(* CODESYS project mqtt_client.20200326.1.project

Project tree, tasks and I/O mapping:
  Device : Changsha-Cyber-MI-linux, Changsha Cyber-MI Co., Ltd., version 3.5.10.40
    application Application
      libraries: Standard, * (System); CAA Memory, 3.5.12.0 (CAA Technical Workgroup); SysTypes2 Interfaces, 3.5.4.0 (System); CAA Net Base Services, 3.5.15.0 (CAA Technical Workgroup); CAA Types Extern, 3.5.13.0 (CAA Technical Workgroup); SysFile, 3.5.15.0 (System); MIC7001 base library, 0.80 (Cyber-MI.com); Util, 3.5.14.0 (System)
      task MainTask (cyclic, interval 10 ms, priority 10, watchdog 200 ms x 1) calls prg_mqtt
      MQTT_Client/
        Function Blocks/
          function block FB_CalculateRemainingLength [ST]
          function block FB_DecodeRemainingLength [ST]
          function block FB_MQTTClient [ST]: m_fill_subscribe_buf, m_fill_publish_buf, m_fill_connect_buf, rm_return, m_read_config
          function block FB_Random [ST]
        Structs/
          data type DUT_json
        Functions/
          function MQTTPacket_encode [ST]
          function MQTTPacket_len [ST]
          function MQTT_connect_len [ST]
          function arr2json [ST]
          function json2arr [ST]
          function get_sub_string [ST]
          function count_char_in_string [ST]
          function rm_left [ST]
      trace Trace (task MainTask): prg_main.rpm_value
      program prg_mqtt [CFC]: ACT_boot, ACT_publish, ACT_recv_proc, ACT_first_buffer, ACT_normal_buffer, ACT_running_light, proc_get_command, proc_set_command, find_key
      global variables GVL
    SoftMotion General Axis Pool
    IoDrvMIC7001 : IoDrvMIC7001, Cyber-MI, version 19.1.1
        output Application.prg_mqtt.led_run : BOOL  // LED_run
        output Application.prg_mqtt.led_err : BOOL  // LED_err
        output Application.prg_mqtt.led_usr : BOOL  // LED_usr
        unmapped channels: Ai00@C16, Ai01@C28, Ai02@C17, Ai03@C29, Ai04@C30, Ai05@C19, Ai06@C31, Ai07@C20, Ai08@C18, Ai09@D18, Ai10@D20, Ai11@D31, Ai12@D19, Ai13@D30, Ai14@D29, Ai15@D17, Ai16@D28, Ai17@D16, Ai18-Do00@C25, Ai19-Do01@C24, Ai20-Do02@C13, Ai21-Do03@C01, Ai22-Do04@C03, Ai23-Do05@C04, Ai24-Do06@C05, Ai25-Do07@C06, Ai26-Do08@C08, Ai27-Do09@C09, Ai28-Do10@C10, Ai29-Do11@C11, Ai30-Do12@D34, Ai31-Do13@D35, Ai32-Do14@D23, Ai33-Do15@D12, Ai34-Do16@D10, Ai35-Do17@D09, Ai36-Do18@D08, Ai37-Do19@D07, Ai38-Do20@D05, Ai39-Do21@D04,
          Ai40-Do22@D03, Ai41-Do23@D02, Ai42-Do24@C23, Ai43-Do25@C35, Ai44-Do26@D24, Ai45-Do27@D13, Ai46-Ao00@C22, Ai47-Ao01@D14, Ai48_Pi02, Ai49_Out5V, Ai50_VCC, Ai51_VCC_L, Ai52_VCC_R, Ai53_Pwm-i0, Ai54_Pwm-i1, Ai55_Pwm-i2, Ai56_Pwm-i3, Ai57_CPU-T, Ai58_G-x, Ai59_G-y, Ai60_G-z, Ai61-reserved, Ai62-IO-cntr, Ai63-CDS-cntr, Di00-Ai00@C16, Di01-Ai01@C28, Di02-Ai02@C17, Di03-Ai03@C29, Di04-Ai04@C30, Di05-Ai05@C19, Di06-Ai06@C31, Di07-Ai07@C20, Di08-Ai08@C18, Di09-Ai09@D18, Di10-Ai10@D20, Di11-Ai11@D31, Di12-Ai12@D19, Di13-Ai13@D30, Di14-Ai14@D29, Di15-Ai15@D17,
          Di16-Ai16@D28, Di17-Ai17@D16, Di18-Ai18@C25, Di19-Ai19@C24, Di20-Ai20@C13, Di21-Ai21@C01, Di22-Ai22@C03, Di23-Ai23@C04, Di24-Ai24@C05, Di25-Ai25@C06, Di26-Ai26@C08, Di27-Ai27@C09, Di28-Ai28@C10, Di29-Ai29@C11, Di30-Ai30@D34, Di31-Ai31@D35, Di32-Ai32@D23, Di33-Ai33@D12, Di34-Ai34@D10, Di35-Ai35@D09, Di36-Ai36@D08, Di37-Ai37@D07, Di38-Ai38@D05, Di39-Ai39@D04, Di40-Ai40@D03, Di41-Ai41@D02, Di42-Ai42@C23, Di43-Ai43@C35, Di44-Ai44@D24, Di45-Ai45@D13, Di46-Ai46@C22, Di47-Ai47@D14, Di48-Pi00@C15, Di49-Pi01@C14, Di50-Pi02@D22, Di51-Pi03@D21, Di52-reserved, Di53-reserved, Di54-reserved, Di55-reserved,
          Di56-reserved, Di57-reserved, Di58-reserved, Di59-reserved, Di60-reserved, Di61-reserved, Di62-reserved, Di63-reserved, Pi00-Di48@C15, Pi01-Di49@C14, Pi02-Di50@D22, Pi03-Di51@D21, Do00-Ai18@C25, Do01-Ai19@C24, Do02-Ai20@C13, Do03-Ai21@C01, Do04-Ai22@C03, Do05-Ai23@C04, Do06-Ai24@C05, Do07-Ai25@C06, Do08-Ai26@C08, Do09-Ai27@C09, Do10-Ai28@C10, Do11-Ai29@C11, Do12-Ai30@D34, Do13-Ai31@D35, Do14-Ai32@D23, Do15-Ai33@D12, Do16-Ai34@D10, Do17-Ai35@D09, Do18-Ai36@D08, Do19-Ai37@D07, Do20-Ai38@D05, Do21-Ai39@D04, Do22-Ai40@D03, Do23-Ai41@D02, Do24-Ai42@C23, Do25-Ai43@C35, Do26-Ai44@D24, Do27-Ai45@D13,
          Do28-Pwmi00@C33, Do29-Pwmi01@C34, Do30-Pwmi02@D25, Do31-Pwmi03@D26, PWM00@C25, PWM01@C24, PWM02@C13, PWM03@C01, PWM04@C03, PWM05@C04, PWM06@C05, PWM07@C06, PWM08@C08, PWM09@C09, PWM10@C10, PWM11@C11, PWM12@D34, PWM13@D35, PWM14@D23, PWM15@D12, PWM16@D10, PWM17@D09, PWM18@D08, PWM19@D07, PWM20@D05, PWM21@D04, PWM22@D03, PWM23@D02, PWM24@C23, PWM25@C35, PWM26@D24, PWM27@D13, PWM28-Pwmi00@C33, PWM29-Pwmi01@C34, PWM30-Pwmi02@D25, PWM31-Pwmi03@D26, PWM_I_0@C33, PWM_I_1@C34, PWM_I_2@D25, PWM_I_3@D26,
          Ao00-Ai46@C22, Ao01-Ai47@D14, ctrl_ai_raw, ctrl_adjust, ctrl_adj0, ctrl_adj1, ctrl_adj2, ctrl_adj3, disable_5V
*)

// Device/Application/MQTT_Client/Structs/DUT_json
TYPE DUT_json :
STRUCT
	key:STRING(32);
	value_dint : DINT;
	value_real : REAL;
	value_str : STRING(128);
	val_tp : UINT;  //0:  int,   1: real,    2: string
END_STRUCT
END_TYPE

// Device/Application/GVL
{attribute 'qualified_only'}

(*start of var_global for mqtt ***************************************************)
VAR_GLOBAL
	xLock_cmd : BOOL := FALSE;
	diLock_grade : DINT := 0;
	diLock_delay : DINT := 0;
	mqtt_interval : DINT := 5;  //mqtt package interval of publish to server
END_VAR

VAR_GLOBAL CONSTANT
	TYPE_DINT:UINT := 0;
	TYPE_REAL:UINT := 1;
	TYPE_STRING:UINT := 2;
END_VAR
(*end of var_global for mqtt *****************************************************)

// Device/Application/prg_mqtt
PROGRAM prg_mqtt

VAR
	FB_MQTTClient_0: FB_MQTTClient;
	
	//topic : STRING(255) := '/sys/a1SB8J9cA4L/CMI010319120011/thing/model/up_raw';
	//topic : STRING(255) := '/a1SB8J9cA4L/CMI010319120011/user/to_app';
	payload : STRING(255) := '{"RPM": 1234, "Hours": 2345}';
	
	//subscribe : STRING(255) := '/a1SB8J9cA4L/CMI010319120011/user/from_app';
	
	xPub : BOOL := FALSE;
	xSub : BOOL := FALSE;
	xBooted :BOOL := FALSE;
	
	ton_pub : ton;
	
	val_payload:ARRAY[0..32] OF dut_json;
	rpm_value : DINT := 1000;
	hours_value :REAL := 680;
	time_value : STRING;
	sn_value : STRING(128);
	lac_str:STRING(128);
	cid_str:STRING(128);
	press_value :REAL := 20.1;
	
	recv_data : ARRAY[0..32] OF DUT_json;
	old_recv_cntr:UDINT := 0;
	payload_len :INT;
	
	mqtt_first :BOOL := TRUE;
	ton_running:ton:=(pt := T#500MS);
	led_run:BOOL := FALSE;
	led_err:BOOL := FALSE;
	led_usr:BOOL := FALSE;
	pkg_id :DINT := 0;
	i :DINT;
END_VAR

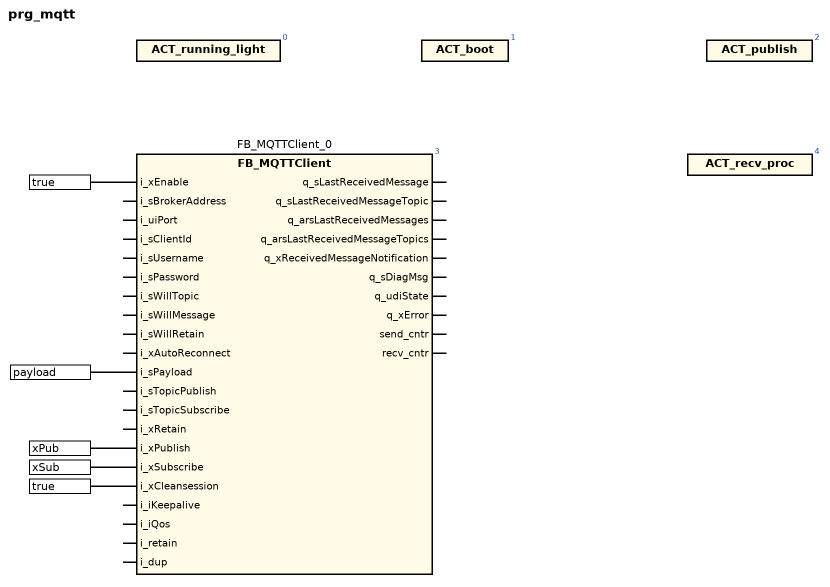
ACT_running_light();
ACT_boot();
ACT_publish();
FB_MQTTClient_0(
    i_xEnable := true,
    i_sPayload := payload,
    i_xPublish := xPub,
    i_xSubscribe := xSub,
    i_xCleansession := true); // FB_MQTTClient
ACT_recv_proc();

ACTION ACT_boot:
IF NOT xbooted THEN
	IF FB_MQTTClient_0.q_udiState = 60 THEN
		FB_MQTTClient_0.i_xSubscribe := TRUE;
		xBooted := TRUE;
	END_IF
END_IF
END_ACTION

ACTION ACT_publish:
IF FB_MQTTClient_0.q_udiState <> 60 THEN   //not ready, return and wait
	xPub := FALSE;
	RETURN;
END_IF

IF mqtt_first THEN
	mqtt_first := FALSE;
	ACT_first_buffer();
	xPub := TRUE;
	RETURN;
END_IF

ton_pub(in := NOT ton_pub.Q, pt := ANY_TO_TIME(gvl.mqtt_interval*1000));   // second to ms
IF ton_pub.Q THEN
	ACT_normal_buffer();
	xPub := TRUE;
ELSE
	xPub := FALSE;
END_IF
END_ACTION

ACTION ACT_recv_proc:
(*
	cmd:  	set, get          			//命令字, set:设置参数或者执行命令，  get：点播数据或参数
	act:  	lock, unlock, reboot		//动作类型
	grade:  1, 2, 3, 4					//动作级别
	delay:  0, 60, 3600					//延迟时间,单位： 秒
*)

IF old_recv_cntr = FB_MQTTClient_0.recv_cntr THEN  //no new message
	RETURN;
END_IF
old_recv_cntr := FB_MQTTClient_0.recv_cntr;

payload_len := json2arr(json := FB_MQTTClient_0.q_sLastReceivedMessage, pArr := ADR(recv_data), max_len := 32);
IF payload_len = 0 THEN
	RETURN;
END_IF

i := find_key(key := 'cmd');
IF i >= 0 AND recv_data[i].val_tp = GVL.TYPE_STRING THEN 
	IF  recv_data[i].value_str = 'get' THEN
		proc_get_command();
	ELSIF recv_data[i].value_str = 'set' THEN
		proc_set_command();
	END_IF
END_IF
END_ACTION

ACTION ACT_first_buffer:

val_payload[0].key := 'sn';
val_payload[0].val_tp := GVL.TYPE_STRING;
IF MIC7001_base.read_sn(ADR(sn_value)) THEN
	val_payload[0].value_str := sn_value;
ELSE
	val_payload[0].value_str := 'SN Error';
END_IF

val_payload[1].key := 'lac';
val_payload[1].val_tp := GVL.TYPE_STRING;

val_payload[2].key := 'cid';
val_payload[2].val_tp := GVL.TYPE_STRING;

IF MIC7001_base.read_location(lac := ADR(lac_str), ci := ADR(cid_str)) THEN
	val_payload[1].value_str := lac_str; 
	val_payload[2].value_str := cid_str; 
ELSE
	val_payload[1].value_str := 'lac_error'; 
	val_payload[2].value_str := 'cid_error'; 
END_IF

payload := arr2json(arr := val_payload, num := 3);
END_ACTION

ACTION ACT_normal_buffer:

val_payload[0].key := 'rpm';
val_payload[0].val_tp := GVL.TYPE_DINT; 
rpm_value := rpm_value + 1;
IF rpm_value > 2200 THEN
	rpm_value := 1000;
END_IF
val_payload[0].value_dint := rpm_value; 

val_payload[1].key := 'hour_all';
val_payload[1].val_tp := GVL.TYPE_REAL;
hours_value := hours_value + 5.0/3600;
val_payload[1].value_real := hours_value; 

val_payload[2].key := 'power';
val_payload[2].val_tp := GVL.TYPE_REAL;  
val_payload[2].value_real := ANY_TO_REAL(rpm_value)/10.0 - 39.0; 

val_payload[3].key := 'press';
val_payload[3].val_tp := GVL.TYPE_REAL;  
press_value := press_value + 0.001;
IF press_value > 35 THEN
	press_value := 20;
END_IF
val_payload[3].value_real := press_value; 

val_payload[4].key := 'fuel_all';
val_payload[4].val_tp := GVL.TYPE_REAL;  
val_payload[4].value_real := ANY_TO_REAL(hours_value)*13.2; 

val_payload[5].key := 'pkg_id';
val_payload[5].val_tp := GVL.TYPE_DINT; 
pkg_id := pkg_id + 1;
val_payload[5].value_dint := pkg_id; 

payload := arr2json(arr := val_payload, num := 6);
END_ACTION

ACTION ACT_running_light:
ton_running(in := NOT ton_running.Q);
IF ton_running.Q THEN
	led_run := NOT led_run;
	led_usr := FALSE;
END_IF

IF FB_MQTTClient_0.q_udiState <> 60 THEN
	led_usr := TRUE;
END_IF
END_ACTION

ACTION proc_get_command:
(*
	cmd:  	get  	//命令字, get：点播数据或参数
	rpm:  	15		//点播转速， 上传15次
	press:  0		//点播压力， 持续上传
	fuel_all: 1	  	//点播总油耗，上传一次 					
*)
END_ACTION

ACTION proc_set_command:
(*
	cmd:  	set  	          	//命令字, set:设置参数或者执行命令，  get：点播数据或参数
	interval:	15				//设置上传间隔： 15秒
	act:  	lock, unlock		//锁机动作类型
	grade:  1, 2, 3, 4			//动作级别
	delay:  0, 60, 3600			//延迟时间,单位： 秒
*)

// check lock command 
i := find_key(key := 'act');
IF i >= 0 AND recv_data[i].val_tp = GVL.TYPE_STRING  THEN
	IF recv_data[i].value_str = 'lock' THEN
		gvl.xlock_cmd := TRUE;
	ELSIF recv_data[i].value_str = 'unlock' THEN
		gvl.xlock_cmd := FALSE;
	END_IF
END_IF

i := find_key(key := 'grade');
IF i >= 0 AND recv_data[i].val_tp = GVL.TYPE_DINT THEN
	gvl.diLock_grade := recv_data[i].value_dint;
END_IF

i := find_key(key := 'delay');
IF i >= 0 AND recv_data[i].val_tp = GVL.TYPE_DINT THEN
	gvl.diLock_delay := recv_data[i].value_dint;
END_IF

i := find_key(key := 'interval');
IF i >= 0 AND recv_data[i].val_tp = GVL.TYPE_DINT THEN
	gvl.mqtt_interval := recv_data[i].value_dint;
END_IF
END_ACTION

METHOD find_key : dint
VAR_INPUT
	key :STRING(32);
END_VAR
VAR
	i :UINT;
END_VAR
find_key := -1;

FOR i := 0 TO payload_len-1 DO
	IF key = recv_data[i].key THEN
		find_key := i;
		RETURN;
	END_IF
END_FOR

RETURN; // not find,  return -1
END_METHOD

END_PROGRAM

// Device/Application/MQTT_Client/Function Blocks/FB_MQTTClient
(*  mqtt client for MIC7001
    by zhoujihui@gmail.com
*)
FUNCTION_BLOCK FB_MQTTClient
VAR_INPUT
	// Enables the Function block, The rising Edge of this Input automatically connects to the MQTT Broker - Standard: TRUE
	i_xEnable: BOOL := TRUE;
	// IP-Address (example: 192.168.178.101) or Webaddress (www.mqtt-dashboard.com) of the MQTT-Broker
	i_sBrokerAddress: STRING(255) := '47.107.240.29';
	// Port of the MQTT-Broker - Standard: 1883
	i_uiPort: UINT := 1883;
	// clientId
	i_sClientId: STRING(255) := 'MIC7001 client Id';
	// Optional Username if required
	i_sUsername: STRING(255) := '';
	// Optional Password if required
	i_sPassword: STRING(255) := '';
	// Last Will Topic if required (Automatically enables Will Message if changed) - otherwise leave untouched
	i_sWillTopic: STRING(255) := '';
	// Last Will Message if required - otherwise leave untouched
	i_sWillMessage: STRING(255) := '';
	// Retain Last Will Message, if required Standard: FALSE - otherwise leave untouched 
	i_sWillRetain: BOOL := FALSE;	
	// Automatically try to reconnect after an Exception - Standard: TRUE
	i_xAutoReconnect: BOOL := TRUE;
	// PayLoad to Publish
	i_sPayload: STRING(255) := '';
	// Topic to Publish to
	i_sTopicPublish: STRING(255) := '/MIC7001/without/config/files';
	// Topic to Subscribe
	i_sTopicSubscribe: STRING(255) := '';
	// Retain Flag Forces the Broker to Retain the Last Mesage - Standard: TRUE
	i_xRetain: BOOL := TRUE;
	// Publish the Payload to the Topic of the MQTT-Broker
	i_xPublish: BOOL:=FALSE;
	// Subscribe to the Topic given to the Input i_sTopicSubscribe
	i_xSubscribe: BOOL:=FALSE;
	// clean session
	i_xCleansession : BOOL := FALSE;
	// keep alive
	i_iKeepalive :INT := 60000;
	// QoS of publish packet
	i_iQos : BYTE := 0;
	// retain
	i_retain : BOOL := FALSE;
	// dup
	i_dup :BOOL := FALSE;
	
END_VAR
VAR_OUTPUT
	// Message Received from a subsribed Topic
	q_sLastReceivedMessage: STRING(255);
	// Topic Message Received
	q_sLastReceivedMessageTopic: STRING(255);	
	// Last 25 Received Messages
	q_arsLastReceivedMessages: STRING(255);
	// Last 25 Topics Received
	q_arsLastReceivedMessageTopics: STRING(255);	
	// Message Received Notification
	q_xReceivedMessageNotification: BOOL;
	// Diag Message
	q_sDiagMsg: STRING(255);
	// Current State of the Function Block
	q_udiState: UDINT;
	// Error Flag
	q_xError: BOOL;
	//publish message counter
	send_cntr :UDINT := 0;
	//received message counter
	recv_cntr: UDINT := 0;
END_VAR
VAR
	R_TRIG_Enable: R_TRIG;

	diResult: CAA.SIZE;
	IFB_CalculateRemainingLength: FB_CalculateRemainingLength;
	IFB_Random: ARRAY[0..9] OF FB_Random;
	wKeepAlive: WORD := 0;
	IoCtlParameter : DINT := 1;

	R_TRIG_Publish: R_TRIG;
	R_TRIG_Subscribe: R_TRIG;

	uiYear:UINT;
	uiMonth: UINT;
	uiDay: UINT;
	uiHour: UINT;
	uiMinute: UINT;
	uiSecond: UINT;
	
	TON_TimeOut: ton;
	wTimeOutValue: WORD;
	udiLastState: UDINT;
	
	xResultDisconnect: BOOL;
	QI: INT;
	
	iIndexCount: INT;
	wPacketIdentifierCount: WORD :=0;
	uiPayLoadLength: uint;
	
	xPublish: BOOL;
	xSubscribe: BOOL;
	
	i: INT;

	hSock:RTS_IEC_HANDLE;
	pSock_create_rst: POINTER TO RTS_IEC_RESULT;
	pSock_recv_rst: POINTER TO RTS_IEC_RESULT;
	pSock_send_rst: POINTER TO RTS_IEC_RESULT;

	ui_rc_disconnect : UDINT;
	pInaddr:POINTER TO STRING;
	
	tcp_client : NBS.TCP_Client;
	tcp_connection : CAA.HANDLE;
	tcp_send : NBS.TCP_Write;
	tcp_recv : NBS.TCP_Read;
	s_send_buf : ARRAY[0..999] OF BYTE;
	s_recv_buf : ARRAY[0..999] OF BYTE;
	udi_time_out : UDINT;
	server_ip : NBS.IP_ADDR;
	buf_size : CAA.size;
	recv_len : INT;

	header :BYTE ; 
	bytes_len_rem : INT;
	length_topic : INT;
	recv_qos : BYTE := 0;
	id_msb : BYTE;
	id_lsb : BYTE;
	hFile: RTS_IEC_HANDLE;
	udiOpenError: RTS_IEC_RESULT;
	udiReadError: RTS_IEC_RESULT;
	str_size: __XWORD;
	udiByteRead: LWORD;	
	str_temp:STRING(255);
	error_cntr : DINT := 0;
END_VAR


R_TRIG_Enable(CLK:=i_xEnable);
R_TRIG_Publish(CLK:=i_xPublish);
R_TRIG_Subscribe(CLK:=i_xSubscribe);

IF (R_TRIG_Publish.Q) THEN
	xPublish:=TRUE;
END_IF

IF (R_TRIG_Subscribe.Q) THEN
	xSubscribe:=TRUE;
END_IF

CASE q_udiState OF
//0: Wait for Enable
0: 	wTimeOutValue:=0;
	
	IF (NOT q_xError) THEN	
		q_sDiagMsg:='Wait for Enable';
	END_IF
	
	IF (i_xEnable OR (i_xAutoReconnect AND q_xError)) THEN
		IF m_read_config() THEN
			q_xError := FALSE;
			q_udiState:=5;
			tcp_client(xEnable := FALSE);
			server_ip.sAddr := i_sBrokerAddress;
			tcp_client.xEnable := TRUE;			
			q_sDiagMsg:='Creating TCP connect';
		ELSE
			q_xError := TRUE;
			q_sDiagMsg:='Failed reading config files';
			q_udiState:=99;
		END_IF
		
	END_IF

5:  
	IF tcp_client.xActive THEN
		q_udiState := 15;
		q_sDiagMsg:='Initialize send-Buffer';
	END_IF
	
	wTimeOutValue:=3000;
	IF (TON_TimeOut.Q) THEN
		q_udiState:=0;	
	END_IF		

//15: Initialize OutBuffer
15:
	buf_size := m_fill_connect_buf();
	IF buf_size > 0 THEN
		tcp_send.szSize := buf_size; 
		tcp_send(xExecute := FALSE);
		tcp_send.xExecute := TRUE;
		tcp_recv.xEnable := TRUE;
		
		q_udiState:=20;
		q_sDiagMsg:='Connect to MQTT-Broker';
	ELSE
		q_xError := TRUE;
		q_sDiagMsg:='Send buffer is Error.';
		q_udiState:=0;
	END_IF
	
//20: Send Connect	
20:		
	wTimeOutValue:=1000;
	tcp_recv(hConnection := tcp_connection, szSize := 1024, pData := ADR(s_recv_buf));
	IF tcp_recv.xReady  THEN
		q_udiState:= 30;
	END_IF
	
	IF (TON_TimeOut.Q) THEN
		q_udiState:=0;	
		q_xError := TRUE;
		q_sDiagMsg:='Connecting to MQTT-Broker (MQTT Control Packet) Timed out';
	END_IF
//30: Analyze CONNACK
30:	q_sDiagMsg:='Analyze connack';
	wTimeOutValue:=0;
	
	IF (s_recv_buf[0] = 32 AND s_recv_buf[3] = 0) THEN
		q_udiState := 60;
	ELSE
		//Return code repsone (2nd Byte): 
		//0: Connection Accepted
		//1: Connection Refused, unacceptable protocol version
		IF (s_recv_buf[3] = 1) THEN
			q_sDiagMsg:='Connection Refused, unacceptable protocol version';
		END_IF
		//2: Connection Refused, identifier rejected
		IF (s_recv_buf[3] = 2) THEN
			q_sDiagMsg:='Connection Refused, identifier rejected';
		END_IF
		//3: Connection Refused, Server unavailable
		IF (s_recv_buf[3] = 3) THEN
			q_sDiagMsg:='Connection Refused, Server unavailable';
		END_IF		
		//4: Connection Refused, bad Username or passworrd
		IF (s_recv_buf[3] = 4) THEN
			q_sDiagMsg:='Connection Refused, bad Username or password';
		END_IF	
		//5: Connection Refused, not autorized
		IF (s_recv_buf[3] = 5) THEN
			q_sDiagMsg:='Connection Refused, not autorized';
		END_IF	
		q_xError := TRUE;
		q_udiState := 90;	
	END_IF
	
//60: Wait for Publish or Disconnect (Enable low)
60:	q_sDiagMsg:='Wait for Publish or Subscribe or Disconnect (Enable low)';
	wTimeOutValue:=0;
	q_xReceivedMessageNotification:= FALSE;

	IF (xPublish) THEN
		xPublish:=FALSE;
		q_udiState := 70;	
	END_IF
	IF (xSubscribe) THEN
		xSubscribe:=FALSE;
		q_udiState := 65;	
	END_IF
	IF (NOT i_xEnable) THEN
		q_udiState := 80;	
	END_IF
	
	tcp_recv(hConnection := tcp_connection, szSize := 1024, pData := ADR(s_recv_buf));
	IF tcp_recv.szCount > 2 THEN
		header := s_recv_buf[0];
		IF header.5 AND header.4 AND tcp_recv.szCount < 1024 THEN   // publish:  0x30
			q_xReceivedMessageNotification:= TRUE;
			diResult := tcp_recv.szCount;
			q_udiState := 63;
			
		END_IF	
	END_IF
	
//Analyze Publish Message from Broker
63: q_sDiagMsg:='Analyze Publish Message from Broker';
	wTimeOutValue:=0;

	IFB_CalculateRemainingLength(wNumberOfBytes:=ANY_TO_WORD(diResult-2));
	bytes_len_rem := IFB_CalculateRemainingLength.iNumberOfBytesRemianingLengthField;
	length_topic := BYTE_TO_INT(s_recv_buf[bytes_len_rem+1])*256 + s_recv_buf[bytes_len_rem+2];
	IF length_topic > 128 THEN
		q_udiState := 60;
		RETURN;	
	END_IF
	
	uiPayLoadLength:=ANY_TO_UINT(diResult - length_topic - 1 - bytes_len_rem - 2);
	header := s_recv_buf[0];
	
	recv_qos := 0;
	IF header.1 OR header.2 THEN //Qos > 0
		uiPayLoadLength :=  uiPayLoadLength - 2;  //remove 2bytes of packet Id
		IF header.1 THEN
			recv_qos := 1;
		ELSIF header.2 THEN
			recv_qos := 2;
		END_IF	

		id_msb := s_recv_buf[1+bytes_len_rem + 2 + length_topic];
		id_lsb := s_recv_buf[1+bytes_len_rem + 2 + length_topic+1];
	END_IF
	
	mem.MemFill(ADR(q_sLastReceivedMessage),255,0);
	mem.MemFill(ADR(q_sLastReceivedMessageTopic),255,0);
	MEM.MemMove(ADR(s_recv_buf[diResult-uiPayLoadLength]),ADR(q_sLastReceivedMessage),uiPayLoadLength);
	MEM.MemMove(ADR(s_recv_buf[IFB_CalculateRemainingLength.iNumberOfBytesRemianingLengthField+3]),ADR(q_sLastReceivedMessageTopic),length_topic);
	
	q_arsLastReceivedMessageTopics:=q_sLastReceivedMessageTopic;
	q_arsLastReceivedMessages:=q_sLastReceivedMessage;
	
	diResult:=0;
	recv_cntr := recv_cntr + 1;
	IF recv_qos = 0 THEN
		q_udiState := 60;
	ELSIF recv_qos = 1 THEN
		
		s_send_buf[0] := 16#40;  //type: puback
		s_send_buf[1] := 2;
		s_send_buf[2] := id_msb;
		s_send_buf[3] := id_lsb;
		tcp_send(xExecute := FALSE);
		tcp_send.xExecute := TRUE;
		tcp_send.szSize := 4;
		q_udiState := 64; // send ack
		wTimeOutValue:=1000;
		q_sDiagMsg:='Send ack to broker';
	ELSE  // qos = 2, not support yet
		q_udiState := 60;
	END_IF	

64:
	IF tcp_send.xDone THEN
		q_udistate := 60;
	END_IF
//65: Subscribe to Topic
65: q_sDiagMsg:='Subscribe to Topic';
	wTimeOutValue:=1000;
	
	buf_size := m_fill_subscribe_buf();
	IF buf_size > 0 THEN
		tcp_send.szSize := buf_size; 
		tcp_send(xExecute := FALSE);
		tcp_send.xExecute := TRUE;
		tcp_recv.xEnable := TRUE;
		q_udiState:=66;	
	ELSE
		q_xError := TRUE;
		q_sDiagMsg:='Subscribe buffer is Error.';
		q_udiState:=0;
	END_IF
	
	tcp_recv(hConnection := tcp_connection, szSize := 1024, pData := ADR(s_recv_buf));
	IF tcp_recv.xDone THEN 
		q_udiState:=66;	
	END_IF	
	IF (TON_TimeOut.Q) THEN
		q_udiState:=90;	
		q_xError := TRUE;
		q_sDiagMsg:='Subscribe (MQTT Control Packet) Timed out';
	END_IF	
	
//66: Wait for SUBACK from Broker
66: //diResult := SysSockRecv(hSocket := hSock,pbyBuffer:=ADR(inBuffer),diBufferSize:=500,diFlags:=0, ADR(pSock_recv_rst));
	q_sDiagMsg:='Wait for SUBACK from Broker';
	wTimeOutValue:=1000;
	tcp_recv(hConnection := tcp_connection, szSize := 1024, pData := ADR(s_recv_buf));
	IF tcp_recv.szCount > 0 THEN
		q_udiState:=67;	
		diResult:=0;
	END_IF
	IF (TON_TimeOut.Q) THEN
		q_udiState:=90;	
		q_xError := TRUE;
		q_sDiagMsg:='Waiting for "Suback" from MQTT-Broker Timed out';
	END_IF

//67: Analyze SUBACK
67:	q_sDiagMsg:='Analyze SUBACK';
	wTimeOutValue:=0;
	tcp_recv(hConnection := tcp_connection, szSize := 1024, pData := ADR(s_recv_buf));
	recv_len := ANY_TO_INT(tcp_recv.szCount);
	IF (s_recv_buf[recv_len-1] < 16#80) THEN
		q_udiState := 60;
		diResult:=0;
	ELSE	
		q_udiState:=90;	
		q_xError := TRUE;
		q_sDiagMsg:='Suback Message reported Failure (Return code 0x80)';
	END_IF
	
//70: Publish Message
70: 
	buf_size := m_fill_publish_buf();

	IF buf_size > 0 THEN
		tcp_send.szSize := buf_size; 
		tcp_send(xExecute := FALSE);
		tcp_send.xExecute := TRUE;
		tcp_recv.xEnable := TRUE;
		q_sDiagMsg:='Publish Message';
		wTimeOutValue:=1000;		
		q_udiState:=75;	
	END_IF
	
75:	
	IF (tcp_send.xDone > 0) THEN 
		q_udiState:=60;	
		send_cntr := send_cntr + 1;
	END_IF	
	IF (TON_TimeOut.Q) THEN
		q_udiState:=90;	
		q_xError := TRUE;
		q_sDiagMsg:='Publishing Message (MQTT Control Packet) Timed out';
	END_IF

//80: Send "Disconnect"
80: s_send_buf[0] := 224;		//MQTT Control Packet Type
	s_send_buf[1] := 0;			//Remaining Length (0)
	tcp_send.szSize := 2;
	tcp_send(xExecute := FALSE);
	tcp_send.xExecute := TRUE;
	
	q_sDiagMsg:='Send Disconnect notification to server';
	wTimeOutValue:=1000;
	q_udiState:=85;

85:	
	IF (tcp_send.xDone) THEN 
		diResult:=0;
		q_udiState:=90;	
	END_IF	
	IF (TON_TimeOut.Q) THEN
		q_udiState:=90;	
		q_xError := TRUE;
		q_sDiagMsg:='Sending Disconnect to MQTT-Broker Timed out';
	END_IF	

//90: Disconnect Socket
90:	tcp_client.xEnable := FALSE;
	IF (NOT q_xError) THEN
		q_sDiagMsg:='Close TCP Socket';
	END_IF
	wTimeOutValue:=1000;
	IF (ui_rc_disconnect = 0) THEN 
		q_udiState:=0;	
	END_IF	
	IF (TON_TimeOut.Q) THEN
		q_udiState:=0;	
		q_xError := TRUE;
		q_sDiagMsg:='Closing TCP-Socket  Timed out';
	END_IF	

99: //error
	wTimeOutValue:=5000;
	IF (TON_TimeOut.Q) THEN
		q_udiState:=0;	
		q_xError := TRUE;
		q_sDiagMsg:='Error status Timed out';
	END_IF	
END_CASE

TON_TimeOut(IN:=(udiLastState=q_udiState) AND (wTimeOutValue <> 0) ,PT:=WORD_TO_TIME(wTimeOutValue));
udiLastState:=q_udiState;

IF q_udiState >= 5 THEN
	tcp_client(xEnable := TRUE, ipAddr := server_ip, uiPort := i_uiPort , udiTimeOut := 0, hConnection => tcp_connection);
	IF tcp_connection > 0 THEN
		tcp_send(udiTimeOut := udi_time_out, hConnection := tcp_connection, pData := ADR(s_send_buf));
	END_IF
END_IF

METHOD m_fill_subscribe_buf : CAA.SIZE
VAR_INPUT
END_VAR

VAR
	i : INT;
	ui_subscribe_len:INT;
	ui_mqtt_msg_len:INT;
	ptr : INT := 0;
	rem_len :INT := 0;
	packet_len : CAA.SIZE := 0;
	rc :INT := 0;
	
	flag :BYTE := 0;
END_VAR
m_fill_subscribe_buf := 0;

ui_subscribe_len := (LEN(i_sTopicSubscribe));

rem_len := ui_subscribe_len + 2 + 2 + 1;  //packet id: 2bytes,  length: 2bytes, QoS: 1byte 
packet_len := MQTTPacket_len(rem_len);

IF packet_len > SIZEOF(s_send_buf) THEN
	m_fill_subscribe_buf := 0;
	RETURN;
END_IF

ptr := 0;
// Header Flag. subscribe command.
flag := 16#82;

IF i_dup THEN
	flag := flag + 8;
END_IF

s_send_buf[ptr] := flag;  ptr := ptr + 1;

// Msg Len.
rc := MQTTPacket_encode(ADR(s_send_buf[ptr]), rem_len);   ptr := ptr + rc;

wPacketIdentifierCount:=wPacketIdentifierCount + 1;
IF (wPacketIdentifierCount = 0) THEN
	wPacketIdentifierCount:=1;
END_IF

// packet id	
s_send_buf[ptr] := UINT_TO_BYTE(wPacketIdentifierCount / 256); ptr := ptr + 1;
s_send_buf[ptr] := UINT_TO_BYTE(wPacketIdentifierCount MOD 256); ptr := ptr + 1;

// topic Length.
s_send_buf[ptr] := UINT_TO_BYTE(ui_subscribe_len / 256); ptr := ptr + 1;
s_send_buf[ptr] := UINT_TO_BYTE(ui_subscribe_len MOD 256); ptr := ptr + 1;

//topic subscribe
FOR i:=0 TO ui_subscribe_len-1 DO
	s_send_buf[ptr] := i_sTopicsubscribe[i]; ptr := ptr + 1;
END_FOR	

s_send_buf[ptr] := i_iQos;

m_fill_subscribe_buf := packet_len;
END_METHOD

METHOD m_fill_publish_buf : CAA.SIZE
VAR_INPUT
END_VAR

VAR
	i : INT;
	ui_client_id_len : INT;
	ui_topic_len :INT;
	ui_payload_len:INT;
	ui_mqtt_msg_len:INT;
	ptr : INT := 0;
	rem_len :INT := 0;
	packet_len : CAA.size := 0;
	rc :INT := 0;
	packet_id : UINT := 1;
	flag :BYTE := 0;
END_VAR
m_fill_publish_buf := 0;

ui_topic_len := (LEN(i_sTopicPublish));
ui_payload_len := (LEN(i_sPayload));

rem_len := ui_topic_len + 2 + ui_payload_len;
IF i_iQos > 0 THEN
	rem_len := rem_len + 2;  // add 2 bytes packet Id
END_IF

packet_len := MQTTPacket_len(rem_len);

IF packet_len > SIZEOF(s_send_buf) THEN
	m_fill_publish_buf := 0;
	RETURN;
END_IF

ptr := 0;
// Header Flag. Publish command.
flag := 16#30;  //publish
IF i_retain THEN
	flag := flag + 1;
END_IF

IF i_iQos > 0 AND i_iQos < 3 THEN
	flag := flag + i_iQos*2;
ELSE
	i_dup := 0;
END_IF

IF i_dup THEN
	flag := flag + 8;
END_IF

s_send_buf[ptr] := flag;  ptr := ptr + 1;

// Msg Len.
rc := MQTTPacket_encode(ADR(s_send_buf[ptr]), rem_len);   ptr := ptr + rc;

//topic
IF ui_topic_len > 0 THEN
	// topic Length.
	s_send_buf[ptr] := UINT_TO_BYTE(ui_topic_len / 256); ptr := ptr + 1;
	s_send_buf[ptr] := UINT_TO_BYTE(ui_topic_len MOD 256); ptr := ptr + 1;
	
	// topic
	FOR i:=0 TO ui_topic_len-1 DO
		s_send_buf[ptr] := i_sTopicPublish[i]; ptr := ptr + 1;
	END_FOR	
END_IF

IF i_iQos > 0 THEN
	wPacketIdentifierCount:=wPacketIdentifierCount + 1;
	IF (wPacketIdentifierCount = 0) THEN
		wPacketIdentifierCount:=1;
	END_IF
	s_send_buf[ptr] := UINT_TO_BYTE(wPacketIdentifierCount / 256); ptr := ptr + 1;
	s_send_buf[ptr] := UINT_TO_BYTE(wPacketIdentifierCount MOD 256); ptr := ptr + 1;
END_IF

//payload
IF ui_payload_len > 0 THEN
	// payload,  no length needed
	FOR i:=0 TO ui_payload_len-1 DO
		s_send_buf[ptr] := i_spayload[i]; ptr := ptr + 1;
	END_FOR	
END_IF

m_fill_publish_buf := packet_len;
END_METHOD

METHOD m_fill_connect_buf : CAA.SIZE
VAR_INPUT
END_VAR

VAR
	ui_client_id_len : INT;	
	ui_username_len : INT;
	ui_password_len : INT;
	ui_will_topic_len : INT;
	ui_will_msg_len : INT;
	ptr:INT := 0;  
	remaining_len :INT;
	packet_len :CAA.SIZE;
	rc :INT;
	flag : BYTE := 0;
END_VAR
m_fill_connect_buf := 0;

ui_client_id_len := (LEN(i_sclientid));
ui_username_len := (LEN(i_sUsername));
ui_password_len := (LEN(i_sPassword));
ui_will_topic_len := (len(i_sWillTopic));
ui_will_msg_len := (len(i_sWillMessage));

remaining_len := MQTT_connect_len(ui_client_id_len, ui_will_topic_len, ui_will_msg_len, ui_username_len, ui_password_len);
packet_len := MQTTPacket_len(remaining_len);

IF packet_len > SIZEOF(s_send_buf) THEN
	m_fill_connect_buf := 0;
	RETURN;
END_IF

ptr := 0;

// Header Flag. Connect command.
s_send_buf[ptr] := 16#10; ptr := ptr + 1;

// Msg Len.
rc := MQTTPacket_encode(ADR(s_send_buf[ptr]), remaining_len);   ptr := ptr + rc;


// Protocal Name Length.
s_send_buf[ptr] := 16#00; ptr := ptr + 1;
s_send_buf[ptr] := 16#04; ptr := ptr + 1;
// Protocal Name.
s_send_buf[ptr] := 16#4D; ptr := ptr + 1;
s_send_buf[ptr] := 16#51; ptr := ptr + 1;
s_send_buf[ptr] := 16#54; ptr := ptr + 1;
s_send_buf[ptr] := 16#54; ptr := ptr + 1;
// Version.
s_send_buf[ptr] := 16#04; ptr := ptr + 1;

// Connect Flags.
flag := 0;
IF i_xCleansession THEN
	flag := flag + 16#02;
END_IF

IF ui_username_len > 0 THEN
	flag := flag + 16#80;
END_IF

IF ui_password_len > 0 THEN
	flag := flag + 16#40;
END_IF

s_send_buf[ptr] := flag;  ptr := ptr + 1;

// Keep Alive.
s_send_buf[ptr] := INT_TO_BYTE(i_iKeepalive / 256); ptr := ptr + 1;
s_send_buf[ptr] := INT_TO_BYTE(i_iKeepalive MOD 256); ptr := ptr + 1;

// Client ID Length.
s_send_buf[ptr] := INT_TO_BYTE(ui_client_id_len / 256); ptr := ptr + 1;
s_send_buf[ptr] := INT_TO_BYTE(ui_client_id_len MOD 256); ptr := ptr + 1;
// Client ID.
FOR i:=0 TO ui_client_id_len-1 DO
	s_send_buf[ptr] := i_sClientId[i]; ptr := ptr + 1;
END_FOR

IF ui_will_topic_len > 0 THEN
	// will topic Length.
	s_send_buf[ptr] := INT_TO_BYTE(ui_will_topic_len / 256); ptr := ptr + 1;
	s_send_buf[ptr] := INT_TO_BYTE(ui_will_topic_len MOD 256); ptr := ptr + 1;
	// will topic.
	FOR i:=0 TO ui_will_topic_len-1 DO
		s_send_buf[ptr] := i_sWilltopic[i]; ptr := ptr + 1;
	END_FOR	
END_IF

IF ui_will_msg_len > 0 THEN
	// will message Length.
	s_send_buf[ptr] := INT_TO_BYTE(ui_will_msg_len / 256); ptr := ptr + 1;
	s_send_buf[ptr] := INT_TO_BYTE(ui_will_msg_len MOD 256); ptr := ptr + 1;
	// will message.
	FOR i:=0 TO ui_will_msg_len-1 DO
		s_send_buf[ptr] := i_sWillmessage[i]; ptr := ptr + 1;
	END_FOR	
END_IF

IF ui_username_len > 0 THEN
	// will message Length.
	s_send_buf[ptr] := INT_TO_BYTE(ui_username_len / 256); ptr := ptr + 1;
	s_send_buf[ptr] := INT_TO_BYTE(ui_username_len MOD 256); ptr := ptr + 1;
	// username
	FOR i:=0 TO ui_username_len-1 DO
		s_send_buf[ptr] := i_susername[i]; ptr := ptr + 1;
	END_FOR	
END_IF

IF ui_password_len > 0 THEN
	// will message Length.
	s_send_buf[ptr] := INT_TO_BYTE(ui_password_len / 256); ptr := ptr + 1;
	s_send_buf[ptr] := INT_TO_BYTE(ui_password_len MOD 256); ptr := ptr + 1;
	// password
	FOR i:=0 TO ui_password_len-1 DO
		s_send_buf[ptr] := i_spassword[i]; ptr := ptr + 1;
	END_FOR	
END_IF


m_fill_connect_buf := packet_len;
END_METHOD

METHOD PRIVATE rm_return : string(255)
VAR_INPUT
	str_in:STRING(255);
END_VAR

VAR
	str_rc:string(255);
	length:INT;
END_VAR
str_rc := str_in;

length := len(str_rc);
IF str_rc[length-1] = 10 THEN   // $N
	str_rc := left(str_rc, length-1);
END_IF

length := len(str_rc);
IF str_rc[length-1] = 10 THEN   // $N
	str_rc := left(str_rc, length-1);
END_IF

length := len(str_rc);
IF str_rc[length-1] = 10 THEN   // $N
	str_rc := left(str_rc, length-1);
END_IF

length := len(str_rc);
IF str_rc[length-1] = 10 THEN   // $N
	str_rc := left(str_rc, length-1);
END_IF

rm_return := str_rc;
END_METHOD

METHOD m_read_config : bool
VAR_INPUT
END_VAR
m_read_config := FALSE;

hFile := sysfileopen(szFile := '/userapp/mqtt_server.txt', am := sysfile.AM_READ, pResult:= ADR(udiOpenError));
IF hFile = RTS_INVALID_HANDLE THEN
	RETURN;
END_IF

//文件存在，开始读取内容
sysfile.SysFileSetPos(hFile:=hFile, ulOffset := 0);
FOR i := 0 TO 255 DO  str_temp[i] := 0; END_FOR
udiByteRead := sysfile.SysFileRead(hfile := hFile,pbyBuffer := ADR(str_temp), ulSize := 250, pResult := ADR(udiReadError));
str_temp := rm_return(str_temp);
IF udiByteRead > 7 THEN  
	i_sBrokerAddress := str_temp;
END_IF
sysfile.SysFileClose(hFile := hFile);	

hFile := sysfileopen(szFile := '/userapp/mqtt_port.txt', am := sysfile.AM_READ, pResult:= ADR(udiOpenError));
IF hFile = RTS_INVALID_HANDLE	THEN
	RETURN;
END_IF
 
//文件存在，开始读取内容
sysfile.SysFileSetPos(hFile:=hFile, ulOffset := 0);
FOR i := 0 TO 255 DO  str_temp[i] := 0; END_FOR
udiByteRead := sysfile.SysFileRead(hfile := hFile,pbyBuffer := ADR(str_temp), ulSize := 32, pResult := ADR(udiReadError));
str_temp := rm_return(str_temp);
IF udiByteRead > 2 THEN  
	i_uiPort := STRING_TO_UINT(str_temp);
END_IF
sysfile.SysFileClose(hFile := hFile);	

hFile := sysfileopen(szFile := '/userapp/mqtt_client_id.txt', am := sysfile.AM_READ, pResult:= ADR(udiOpenError));
IF hFile = RTS_INVALID_HANDLE	THEN
	RETURN;
END_IF 
//文件存在，开始读取内容
sysfile.SysFileSetPos(hFile:=hFile, ulOffset := 0);
FOR i := 0 TO 255 DO  str_temp[i] := 0; END_FOR
udiByteRead := sysfile.SysFileRead(hfile := hFile,pbyBuffer := ADR(str_temp), ulSize := 250, pResult := ADR(udiReadError));
str_temp := rm_return(str_temp);
IF udiByteRead > 7 THEN  
	i_sClientId := str_temp;
END_IF
sysfile.SysFileClose(hFile := hFile);	

hFile := sysfileopen(szFile := '/userapp/mqtt_username.txt', am := sysfile.AM_READ, pResult:= ADR(udiOpenError));
IF hFile = RTS_INVALID_HANDLE	THEN
	RETURN;
END_IF
 
//文件存在，开始读取内容
sysfile.SysFileSetPos(hFile:=hFile, ulOffset := 0);
FOR i := 0 TO 255 DO  str_temp[i] := 0; END_FOR
udiByteRead := sysfile.SysFileRead(hfile := hFile,pbyBuffer := ADR(str_temp), ulSize := 250, pResult := ADR(udiReadError));
str_temp := rm_return(str_temp);
IF udiByteRead > 7 THEN  
	i_sUsername := str_temp;
END_IF
sysfile.SysFileClose(hFile := hFile);	

hFile := sysfileopen(szFile := '/userapp/mqtt_password.txt', am := sysfile.AM_READ, pResult:= ADR(udiOpenError));
IF hFile = RTS_INVALID_HANDLE	THEN
	RETURN;
END_IF 
//文件存在，开始读取内容
sysfile.SysFileSetPos(hFile:=hFile, ulOffset := 0);
FOR i := 0 TO 255 DO  str_temp[i] := 0; END_FOR
udiByteRead := sysfile.SysFileRead(hfile := hFile,pbyBuffer := ADR(str_temp), ulSize := 250, pResult := ADR(udiReadError));
str_temp := rm_return(str_temp);
IF udiByteRead > 7 THEN
	i_sPassword := str_temp;
END_IF
sysfile.SysFileClose(hFile := hFile);	

hFile := sysfileopen(szFile := '/userapp/mqtt_topic_publish.txt', am := sysfile.AM_READ, pResult:= ADR(udiOpenError));
IF hFile = RTS_INVALID_HANDLE	THEN
	RETURN;
END_IF
 
//文件存在，开始读取内容
sysfile.SysFileSetPos(hFile:=hFile, ulOffset := 0);
FOR i := 0 TO 255 DO  str_temp[i] := 0; END_FOR
udiByteRead := sysfile.SysFileRead(hfile := hFile,pbyBuffer := ADR(str_temp), ulSize := 250, pResult := ADR(udiReadError));
str_temp := rm_return(str_temp);
IF udiByteRead > 7 THEN
	i_sTopicPublish := str_temp;
END_IF
sysfile.SysFileClose(hFile := hFile);	

hFile := sysfileopen(szFile := '/userapp/mqtt_topic_subscribe.txt', am := sysfile.AM_READ, pResult:= ADR(udiOpenError));
IF hFile = RTS_INVALID_HANDLE	THEN
	RETURN;
END_IF
 
//文件存在，开始读取内容
sysfile.SysFileSetPos(hFile:=hFile, ulOffset := 0);
FOR i := 0 TO 255 DO  str_temp[i] := 0; END_FOR
udiByteRead := sysfile.SysFileRead(hfile := hFile,pbyBuffer := ADR(str_temp), ulSize := 250, pResult := ADR(udiReadError));
str_temp := rm_return(str_temp);
IF udiByteRead > 7 THEN  
	i_sTopicSubscribe := str_temp;
END_IF
sysfile.SysFileClose(hFile := hFile);	

m_read_config := TRUE;
END_METHOD

END_FUNCTION_BLOCK

// Device/Application/MQTT_Client/Function Blocks/FB_CalculateRemainingLength
{attribute 'hide'}
FUNCTION_BLOCK FB_CalculateRemainingLength
VAR_INPUT
	wNumberOfBytes: WORD;
	
END_VAR
VAR_OUTPUT
	iNumberOfBytesRemianingLengthField: INT;
	arbyRemainingBytesField: ARRAY[0..3] OF BYTE;
END_VAR
VAR
	bEncodedByte: BYTE;
	wValue: WORD;
	iCount: INT;
END_VAR

wValue:=wNumberOfBytes;
iCount := 0;
REPEAT
	bEncodedByte:=UINT_TO_BYTE(wValue MOD 128);
	wValue:=wVALUE / 128;
	
	IF (wVALUE > 0) THEN
		bEncodedByte := (bEncodedByte AND 128);
	END_IF
	arbyRemainingBytesField[iCount] := bEncodedByte;
	iCount := iCount + 1;

UNTIL (wValue <= 0)
END_REPEAT;
iNumberOfBytesRemianingLengthField:=iCount;

END_FUNCTION_BLOCK

// Device/Application/MQTT_Client/Function Blocks/FB_Random
	{attribute 'hide'}
FUNCTION_BLOCK FB_Random
VAR_INPUT
	A: DWORD;
	B: DWORD;
	V: DWORD;
END_VAR
VAR_OUTPUT
	dwRandom: dword;
END_VAR
VAR
	dwValue1: DWORD;
	dwValue2: DWORD;
	M: DWORD;
	Q: DWORD;

END_VAR


Q:=Q+2;

M:=25;
dwRandom:=(A+V+B+Q) MOD M + 65;

END_FUNCTION_BLOCK

// Device/Application/MQTT_Client/Functions/MQTTPacket_len
FUNCTION MQTTPacket_len : CAA.SIZE
VAR_INPUT
	rem_len:INT;
END_VAR
VAR
END_VAR


rem_len := rem_len + 1; (* header byte *)

(* now remaining_length field *)
IF rem_len < 128 THEN
   rem_len := rem_len + 1;
ELSIF rem_len < 16384 THEN
   rem_len := rem_len + 2;
ELSIF rem_len < 2097151 THEN
   rem_len := rem_len + 3;
ELSE
   rem_len := rem_len + 4;
END_IF

MQTTPacket_len := rem_len;
RETURN;

END_FUNCTION

// Device/Application/MQTT_Client/Functions/MQTTPacket_encode
FUNCTION MQTTPacket_encode : INT
VAR_INPUT
	buf:POINTER TO BYTE;
	length : INT;
END_VAR
VAR
	rc : INT := 0;
	d : BYTE;
END_VAR


rc := 0;

WHILE length > 0  DO
	d := ANY_TO_BYTE(length MOD 128);
	length := length / 128;
	IF length > 0 THEN
		d := d + 16#80;
	END_IF
	buf[rc] := d;
	rc := rc + 1;
END_WHILE

MQTTPacket_encode := rc;

END_FUNCTION

// Device/Application/MQTT_Client/Functions/MQTT_connect_len
FUNCTION MQTT_connect_len : INT
VAR_INPUT
	len_clientId : INT;
	len_will_topic : INT;
	len_will_msg : INT;
	len_username : INT;
	len_password : INT;
END_VAR
VAR
	len :INT;
END_VAR


len := 10;  //  version 4

len := len + len_clientId + 2;

IF len_will_topic > 0 THEN
	len := len + len_will_topic + 2 + len_will_msg + 2;
END_IF

IF len_username > 0 THEN
	len := len + len_username + 2;
END_IF

IF len_password > 0 THEN
	len := len + len_password + 2;
END_IF


MQTT_connect_len := len;

END_FUNCTION

// Device/Application/MQTT_Client/Functions/json2arr
FUNCTION json2arr : INT
VAR_INPUT
	json : STRING(256);
	pArr : POINTER TO DUT_json;
	max_len : UINT;
END_VAR
VAR
	length : INT;  //length of json string
	number : INT;
	n : INT; 
	p :POINTER TO DUT_json;
	sj : STRING(255);
	str_val : STRING(255);
	
	kv:ARRAY[0..32] OF STRING(255);
	char_l : STRING(1);
	char_r : STRING(1);
	kv_str: STRING(255);
	pos : INT;
END_VAR

//将json格式的字符串分解为结构数组，当前支持的数据类型有： 整型、浮点型、字符串。 键值必须是字符串，并且不支持嵌套

json2arr := 0;

//check format
sj := json;
length := len(sj);
IF length < 7 THEN
	RETURN;
END_IF

n := count_char_in_string(sj, '{');
IF n <> 1 THEN
	RETURN;
END_IF

n := count_char_in_string(sj, '}');
IF n <> 1 THEN
	RETURN;
END_IF

n := count_char_in_string(sj, ',');

number := count_char_in_string(sj, ':');
IF number = 0 THEN
	RETURN;
END_IF

IF number - n <> 1 THEN  // ':'s are more 1 than ','
	RETURN;
END_IF

//split json to array of kv string
FOR n := 0 TO number - 1 DO
	char_l := ',';
	char_r := ',';
	IF n = 0 THEN
		char_l := '{';
	ELSIF n = number -1 THEN
		char_r := '}';
	END_IF
	kv[n] := get_sub_string(sj, char_l, char_r);
	sj := rm_left(sj, '"');  //remove '{' or ',' at the start of current string
	sj := rm_left(sj, char_r); //remove the first key-value
END_FOR

//split key and value, and move to recv_data which is pointed by pArr
FOR n := 0 TO number - 1 DO
	kv_str := kv[n];
	pos := find(kv_str, ':'); 
	IF  pos < 1 THEN  //error
		RETURN;
	END_IF
	
	pArr[n].key := get_sub_string(kv_str, '"', '"');
	str_val := get_sub_string(kv_str, ':', '&');

	IF find(str_val, '"') > 0 THEN //string
		pArr[n].val_tp := 2;
		pArr[n].value_str := get_sub_string(str_val, '"', '"');
	ELSIF find(str_val, '.') > 0 THEN //real
		pArr[n].val_tp := 1;
 		pArr[n].value_real := STRING_TO_REAL(str_val);
	ELSE
		pArr[n].val_tp := 0;
 		pArr[n].value_dint := STRING_TO_DINT(str_val);
	END_IF
		
END_FOR

json2arr := number;

END_FUNCTION

// Device/Application/MQTT_Client/Functions/count_char_in_string
FUNCTION count_char_in_string : int
VAR_INPUT
	in_str : STRING(255);
	ch : STRING(1);
END_VAR
VAR
	cnt : INT := 0;
	pos : INT;
	temp_str : STRING(255);
END_VAR



temp_str := in_str;

cnt := 0;
pos := find(temp_str, ch);
IF pos > 0 THEN
	cnt := cnt + 1;
END_IF

WHILE pos > 0 DO
	temp_str := right(temp_str, len(temp_str)-pos);
	pos := find(temp_str, ch);
	IF pos > 0 THEN
		cnt := cnt + 1;
	END_IF	
END_WHILE

count_char_in_string := cnt;

END_FUNCTION

// Device/Application/MQTT_Client/Functions/get_sub_string
FUNCTION get_sub_string : string(255)
VAR_INPUT
	in_str : STRING(255);
	char_l : STRING(1);
	char_r : STRING(1);
END_VAR
VAR
	start : INT;
	end : INT;
	sub_str : STRING(255);
	length : INT;
END_VAR

get_sub_string := '';

length := len(in_str);
start := 0;
end := length+1;

start := find(in_str, char_l);
sub_str := right(in_str, length-start);
length := len(sub_str);
end := find(sub_str, char_r);
IF end = 0 THEN
	end := length + 1;
END_IF
get_sub_string := left(sub_str, end-1);

END_FUNCTION

// Device/Application/MQTT_Client/Functions/rm_left
FUNCTION rm_left : string(255)
VAR_INPUT
	str_in:STRING(255);
	ch : string(1);
END_VAR
VAR
	pos : INT;
END_VAR


//删除字符串中特定字符左侧的部分，该字符保留。 如果没有发现该指定字符，则返回原字符串
rm_left := str_in;

pos := find(str_in, ch);
IF pos < 0 THEN
	RETURN; 
END_IF

rm_left := right(str_in, len(str_in)-pos+1);

END_FUNCTION

// Device/Application/MQTT_Client/Functions/arr2json
FUNCTION arr2json : string(255)
VAR_INPUT
	arr:ARRAY[0..32] OF dut_json;
	num : INT;
END_VAR
VAR
	i :INT;
	kv : DUT_json;
END_VAR


arr2json := '{';
FOR i := 0 TO num -1 DO
	kv := arr[i];
	arr2json := concat(arr2json, '"');
	arr2json := concat(arr2json, kv.key);
	arr2json := concat(arr2json, '":');
	IF kv.val_tp = GVL.TYPE_DINT THEN   
		arr2json := concat(arr2json, DINT_TO_STRING(kv.value_dint));		
	ELSIF kv.val_tp = GVL.TYPE_REAL THEN  
		arr2json := concat(arr2json, REAL_TO_STRING(kv.value_real));
	ELSIF kv.val_tp = GVL.TYPE_STRING THEN  
		arr2json := concat(arr2json, '"');
		arr2json := concat(arr2json, kv.value_str);
		arr2json := concat(arr2json, '"');	
	ELSE
		arr2json := 'Error:  Value type is unknow.';
		RETURN;	
	END_IF
	IF i <> num-1 THEN
		arr2json := concat(arr2json, ',');
	END_IF
END_FOR

arr2json := concat(arr2json, '}');

END_FUNCTION

// Device/Application/MQTT_Client/Function Blocks/FB_DecodeRemainingLength
FUNCTION_BLOCK FB_DecodeRemainingLength
VAR_INPUT
	abyRemainingLengthField: ARRAY[0..3] OF BYTE;
END_VAR
VAR_OUTPUT
	uiRemeiningLength: UINT;
END_VAR
VAR
	multiplier: UINT;
	value: UINT;
	iCount: INT;
END_VAR

multiplier := 1;
value := 0;
iCount :=0;
REPEAT
	value := value + (abyRemainingLengthField [iCount] AND 127)*multiplier;
	multiplier := multiplier * 128;
UNTIL ((abyRemainingLengthField [iCount] AND 128) <> 0)
END_REPEAT;
uiRemeiningLength:=value;

END_FUNCTION_BLOCK
